// TIA Portal V15.1 export
// export: Created 2020-06-12T07:35:54.2724609Z, ExportSetting None, DisplayName Totally Integrated Automation Portal, DisplayVersion V15.1, DisplayName TIA Portal Openness, DisplayVersion V15.1, DisplayName STEP 7 Professional, DisplayVersion V15.1, DisplayName STEP 7 Safety, DisplayVersion V15.1, DisplayName WinCC Advanced, DisplayVersion V15.1
FUNCTION "Desk_ES1GD01" : Void   // FC162, FBD
{ S7_Optimized_Access := 'TRUE' }
// stored: SetENOAutomatically False
   VAR_TEMP
      FL_DeskActive : Bool;
      FL_Electrodes1_3_man : Bool;
      FL_Electrode1_man : Bool;
      FL_Electrode2_man : Bool;
      FL_Electrode3_man : Bool;
      tHorn : Bool;
      tbool : Bool;
   END_VAR
BEGIN

REGION Network 1: ******************** Control Desk imputs and indicators ******************************
END_REGION

REGION Network 2: ES1GD01_S16_ltest - ES1GD01 PB Lamp test
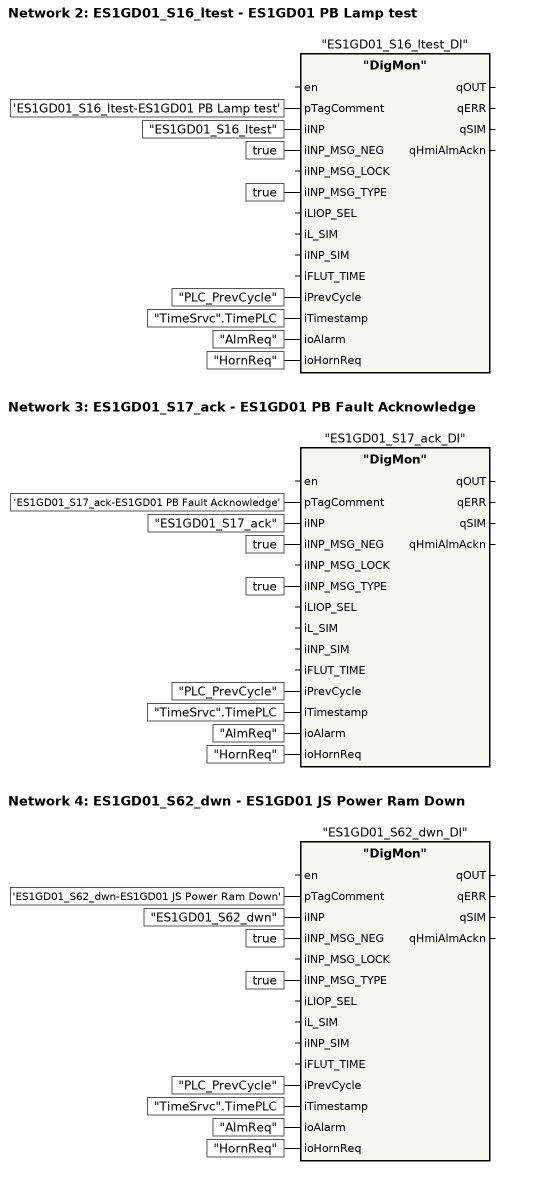
   "ES1GD01_S16_ltest_DI"(pTagComment := 'ES1GD01_S16_ltest-ES1GD01 PB Lamp test',   // "DigMon"
                          iINP := "ES1GD01_S16_ltest",
                          iINP_MSG_NEG := true,
                          iINP_MSG_TYPE := true,
                          iPrevCycle := "PLC_PrevCycle",
                          iTimestamp := "TimeSrvc".TimePLC,
                          ioAlarm := "AlmReq",
                          ioHornReq := "HornReq");
END_REGION

REGION Network 3: ES1GD01_S17_ack - ES1GD01 PB Fault Acknowledge
   "ES1GD01_S17_ack_DI"(pTagComment := 'ES1GD01_S17_ack-ES1GD01 PB Fault Acknowledge',   // "DigMon"
                        iINP := "ES1GD01_S17_ack",
                        iINP_MSG_NEG := true,
                        iINP_MSG_TYPE := true,
                        iPrevCycle := "PLC_PrevCycle",
                        iTimestamp := "TimeSrvc".TimePLC,
                        ioAlarm := "AlmReq",
                        ioHornReq := "HornReq");
END_REGION

REGION Network 4: ES1GD01_S62_dwn - ES1GD01 JS Power Ram Down
   "ES1GD01_S62_dwn_DI"(pTagComment := 'ES1GD01_S62_dwn-ES1GD01 JS Power Ram Down',   // "DigMon"
                        iINP := "ES1GD01_S62_dwn",
                        iINP_MSG_NEG := true,
                        iINP_MSG_TYPE := true,
                        iPrevCycle := "PLC_PrevCycle",
                        iTimestamp := "TimeSrvc".TimePLC,
                        ioAlarm := "AlmReq",
                        ioHornReq := "HornReq");
END_REGION

REGION Network 5: ES1GD01_S62_f - ES1GD01 JS Power Ram Fast
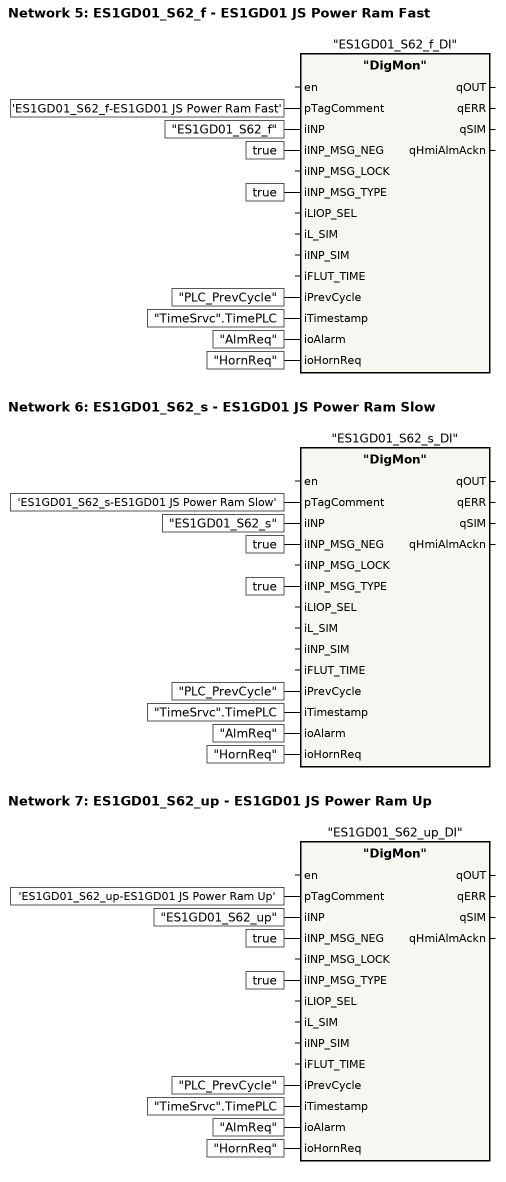
   "ES1GD01_S62_f_DI"(pTagComment := 'ES1GD01_S62_f-ES1GD01 JS Power Ram Fast',   // "DigMon"
                      iINP := "ES1GD01_S62_f",
                      iINP_MSG_NEG := true,
                      iINP_MSG_TYPE := true,
                      iPrevCycle := "PLC_PrevCycle",
                      iTimestamp := "TimeSrvc".TimePLC,
                      ioAlarm := "AlmReq",
                      ioHornReq := "HornReq");
END_REGION

REGION Network 6: ES1GD01_S62_s - ES1GD01 JS Power Ram Slow
   "ES1GD01_S62_s_DI"(pTagComment := 'ES1GD01_S62_s-ES1GD01 JS Power Ram Slow',   // "DigMon"
                      iINP := "ES1GD01_S62_s",
                      iINP_MSG_NEG := true,
                      iINP_MSG_TYPE := true,
                      iPrevCycle := "PLC_PrevCycle",
                      iTimestamp := "TimeSrvc".TimePLC,
                      ioAlarm := "AlmReq",
                      ioHornReq := "HornReq");
END_REGION

REGION Network 7: ES1GD01_S62_up - ES1GD01 JS Power Ram Up
   "ES1GD01_S62_up_DI"(pTagComment := 'ES1GD01_S62_up-ES1GD01 JS Power Ram Up',   // "DigMon"
                       iINP := "ES1GD01_S62_up",
                       iINP_MSG_NEG := true,
                       iINP_MSG_TYPE := true,
                       iPrevCycle := "PLC_PrevCycle",
                       iTimestamp := "TimeSrvc".TimePLC,
                       ioAlarm := "AlmReq",
                       ioHornReq := "HornReq");
END_REGION

REGION Network 8: ES1GD01_S62_zero - ES1GD01 JS Power Ram no movement
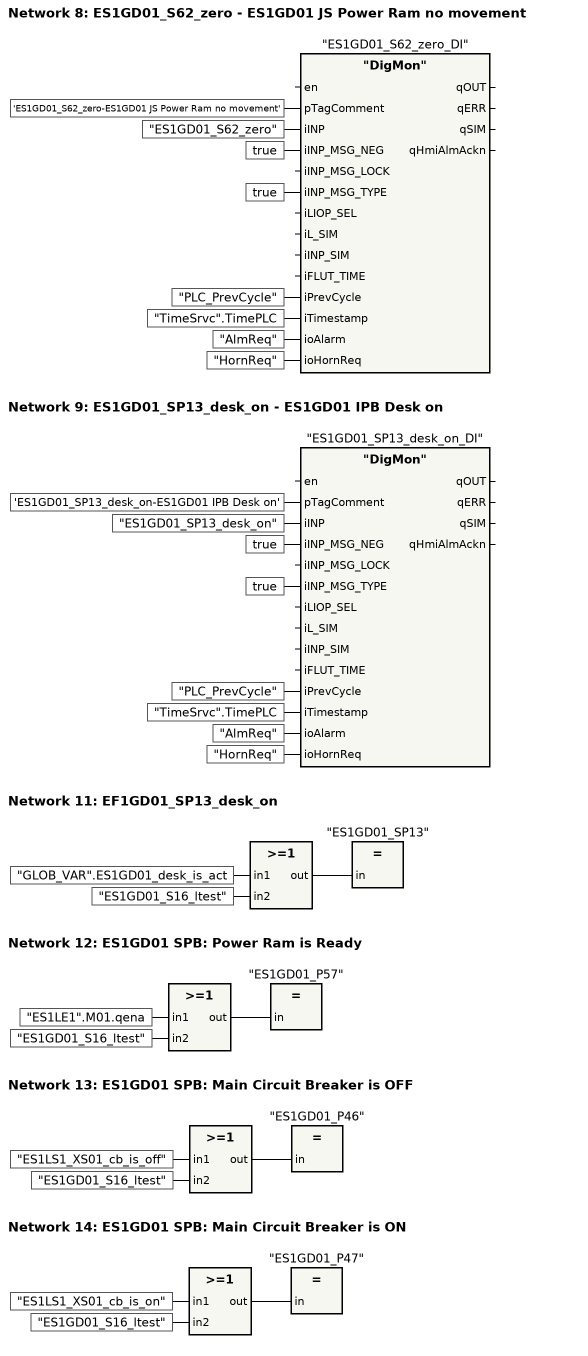
   "ES1GD01_S62_zero_DI"(pTagComment := 'ES1GD01_S62_zero-ES1GD01 JS Power Ram no movement',   // "DigMon"
                         iINP := "ES1GD01_S62_zero",
                         iINP_MSG_NEG := true,
                         iINP_MSG_TYPE := true,
                         iPrevCycle := "PLC_PrevCycle",
                         iTimestamp := "TimeSrvc".TimePLC,
                         ioAlarm := "AlmReq",
                         ioHornReq := "HornReq");
END_REGION

REGION Network 9: ES1GD01_SP13_desk_on - ES1GD01 IPB Desk on
   "ES1GD01_SP13_desk_on_DI"(pTagComment := 'ES1GD01_SP13_desk_on-ES1GD01 IPB Desk on',   // "DigMon"
                           iINP := "ES1GD01_SP13_desk_on",
                           iINP_MSG_NEG := true,
                           iINP_MSG_TYPE := true,
                           iPrevCycle := "PLC_PrevCycle",
                           iTimestamp := "TimeSrvc".TimePLC,
                           ioAlarm := "AlmReq",
                           ioHornReq := "HornReq");
END_REGION

REGION Network 11: EF1GD01_SP13_desk_on
   "ES1GD01_SP13" := "GLOB_VAR".ES1GD01_desk_is_act OR "ES1GD01_S16_ltest";
END_REGION

REGION Network 12: ES1GD01 SPB: Power Ram is Ready
   "ES1GD01_P57" := "ES1LE1".M01.qena OR "ES1GD01_S16_ltest";
END_REGION

REGION Network 13: ES1GD01 SPB: Main Circuit Breaker is OFF
   "ES1GD01_P46" := "ES1LS1_XS01_cb_is_off" OR "ES1GD01_S16_ltest";
END_REGION

REGION Network 14: ES1GD01 SPB: Main Circuit Breaker is ON
   "ES1GD01_P47" := "ES1LS1_XS01_cb_is_on" OR "ES1GD01_S16_ltest";
END_REGION

REGION Network 15: ES1GD01 SPB: Control Voltage ON
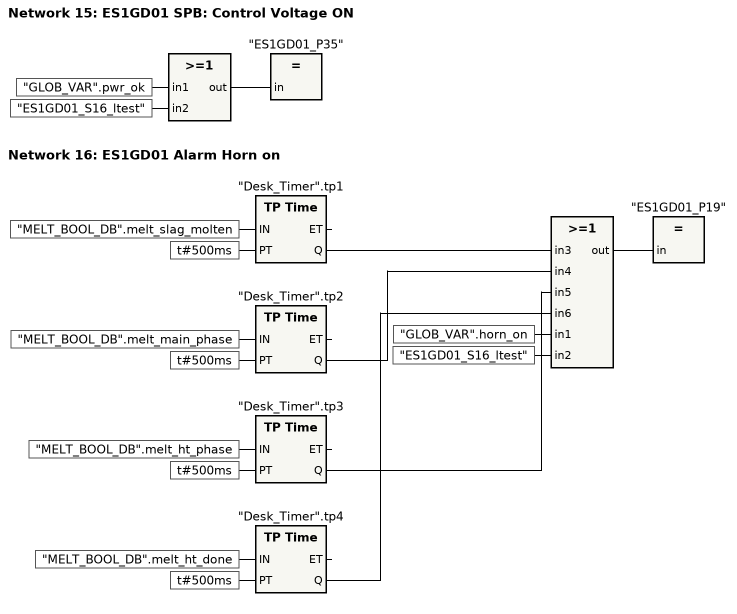
   "ES1GD01_P35" := "GLOB_VAR".pwr_ok OR "ES1GD01_S16_ltest";
END_REGION

REGION Network 16: ES1GD01 Alarm Horn on
   "Desk_Timer".tp1.TP(IN := "MELT_BOOL_DB".melt_slag_molten, PT := t#500ms);
   "Desk_Timer".tp2.TP(IN := "MELT_BOOL_DB".melt_main_phase, PT := t#500ms);
   "Desk_Timer".tp3.TP(IN := "MELT_BOOL_DB".melt_ht_phase, PT := t#500ms);
   "Desk_Timer".tp4.TP(IN := "MELT_BOOL_DB".melt_ht_done, PT := t#500ms);
   "ES1GD01_P19" := "Desk_Timer".tp1.Q OR "Desk_Timer".tp2.Q OR "Desk_Timer".tp3.Q OR "Desk_Timer".tp4.Q OR "GLOB_VAR".horn_on OR "ES1GD01_S16_ltest";
END_REGION
END_FUNCTION
